{attribute 'qualified_only'}
VAR_GLOBAL	
	Inicio_calibracion			:BOOL;
	Pausa_calibracion			:BOOL;
	VaciarProbeta_calibracion	:BOOL;//probeta llena	
	Fin_calibracion				:BOOL;
	Error_promedio				:REAL;
	Continuar_calibracion		:BOOL;
	Volumen_calibracion			:ARRAY[1..3]OF REAL;
	Tiempo_calibracion			:ARRAY[1..3]OF DINT;
	Peso_calibracion			:REAL;
	Dosis_calibracion			:REAL;
	VolumenPedido_calibracion	:REAL;
	Tolerancia_calibracion		:REAL;
	TInyeccion_calibracion		:DINT;
	VolMaxProbeta_calibracion	:REAL;
	Vol_enProbeta				:REAL;
	TiempoInyectado				:DINT;
END_VAR

(* stored: Version 1.1.0.1, ProductVersion 3.1.4024.14
   GVL HMICA2: Id {ede3844a-944b-43ca-9d5f-82dcd67f5c06} *)
